Fanuc KAREL source: ka00143.KL

-- PROVISIONAL review KL for V940-1; original PC SHA256 769cb563f7aa32678d862b9efef8ff07fa2012a1f4d76b58b4ba74ae18d2f164
-- Incomplete behavior may be omitted. Consult companion uncertainty JSON. Do not deploy.
PROGRAM KA00143
%NOLOCKGROUP
-- UNRESOLVED_DECL SRC type=002017
-- UNRESOLVED_DECL DST type=002018
BEGIN
  -- V9_ZERO_TABLE_METADATA_HINT layout=0001; no indexed target words; source/name/runtime held
  -- UNRESOLVED_PC offsets 5-19; opcodes 2E,22,9D,33,B4
  -- UNRESOLVED_PC offsets 24-42; opcodes 22,9D,33,B3,22,9D,33,B2
  -- UNRESOLVED_PC offsets 47-51; opcodes 7F
END KA00143
